INTERFACE IN2PurgeBlock

PROPERTY pEndFeedback : BOOL
GET
END_GET
END_PROPERTY

METHOD Purge : BOOL
VAR_INPUT
	bStartCommand : BOOL;
	sSourceName : STRING;
	nCurrentBlock : INT;	
END_VAR
END_METHOD

END_INTERFACE

(* stored: Version 1.1.0.1, ProductVersion 3.1.4024.9
   Itf IN2PurgeBlock: Id {49d1b0c2-3067-479a-a521-bdd3c054b50f}
   Property pEndFeedback: Id {2f750d42-8df2-4412-a0cd-03c6c0567e08}
   Get Get: Id {58d855c7-e58d-4c96-a9e6-ad9c0140fdd0}
   Method Purge: Id {a215b1dd-2df2-4e07-81f8-175737f3eddc} *)
